(* IEC 61131-3 sources: plc_simulator/services/codesys/POUs (part 9) *)

(* ---- STC_FB_Calibrate.st ---- *)
(* ============================================================
   STC_FB_Calibrate — Teaching / calibration mode
   ============================================================
   Runs 2 normal tasks per transporter to measure real lift,
   sink, and travel kinematic parameters.

   Task 1: lift=dry_station, sink=wet_station
     → MeasureMoveTimes records: lift_s[dry], sink_s[wet],
       travel[dry→wet]
     → X velocity profile measured during phase 3.

   Task 2: lift=wet_station, sink=dry_station
     → MeasureMoveTimes records: lift_s[wet], sink_s[dry],
       travel[wet→dry]

   Two tasks give ALL measurements: lift_wet, sink_wet,
   lift_dry, sink_dry, and X kinematics from vel profile.

   Calibration sequence per transporter:
     Step 10-12: Task 1 (dry→wet) + X velocity measurement
     Step 20-22: Task 2 (wet→dry)
     Step 30:    Read results from g_move → g_cal
     Step 40:    Next transporter or cal_step 100

   Global control:
     Step   0: Idle (waiting for cmd=1)
     Step 100: All measurement done (waiting for cmd=2 = Calculate)
     Step 200: Calculating g_move from measured parameters
     Step 999: Complete (waiting for cmd=3 = abort/reset)

   Inputs:
     i_run  — enable (typically init_done)
     i_cmd  — one-shot command: 1=start, 2=calculate, 3=abort

   Outputs:
     o_step   — current cal_step number
     o_tid    — transporter being calibrated
     o_active — TRUE while calibration is running
   ============================================================ *)

FUNCTION_BLOCK STC_FB_Calibrate
VAR_INPUT
  i_run : BOOL;       (* enable — typically init_done *)
  i_cmd : INT;        (* one-shot: 1=start, 2=calculate, 3=abort *)
END_VAR
VAR_OUTPUT
  o_step   : INT;     (* current calibration cal_step *)
  o_tid    : INT;     (* transporter being calibrated *)
  o_active : BOOL;    (* calibration in progress *)
END_VAR
VAR_EXTERNAL CONSTANT
    MAX_Transporters    : INT;
    MIN_StationIndex : INT;
    MAX_StationIndex   : INT;
END_VAR

VAR_EXTERNAL
  g_transporter : ARRAY[1..MAX_Transporters] OF UDT_TransporterStatusType;
  g_sim_trans   : ARRAY[1..MAX_Transporters] OF UDT_JC_SimTransporterType;
  g_station    : ARRAY[MIN_StationIndex..MAX_StationIndex] OF UDT_StationType;
  g_cfg         : ARRAY[1..MAX_Transporters] OF UDT_TransporterType;
  g_cal         : ARRAY[1..MAX_Transporters] OF UDT_JC_CalibrationType;
  g_move        : ARRAY[1..MAX_Transporters] OF UDT_JC_MoveTimesType;
  g_time_s      : LINT;
END_VAR
VAR
  cal_step       : INT := 0;
  tid        : INT := 0;      (* current transporter 1..3 *)
  task_key   : LINT := 0;   (* task_id for issued task *)
  (* X velocity measurement during phase 3 of task 1 *)
  x_meas_ph  : INT := 0;      (* 0=wait 1=accel 2=cruise 3=decel *)
  x_timer    : REAL := 0.0;
  x_prev_v   : REAL := 0.0;
  x_max_v    : REAL := 0.0;
  x_acc_t    : REAL := 0.0;
  x_dec_t    : REAL := 0.0;
  cur_v      : REAL;
  (* Calculation loop variables *)
  ci         : INT;
  cj         : INT;
  dist       : REAL;
  d_acc      : REAL;
  d_dec      : REAL;
  v_peak     : REAL;
  travel_t   : REAL;
  vm         : REAL;
  ta         : REAL;
  td         : REAL;
  (* Helper *)
  next_tid   : INT;
  wet_idx    : INT;
  dry_idx    : INT;
END_VAR

IF NOT i_run THEN
  RETURN;
END_IF;

(* ── Command handling ── *)
IF i_cmd = 1 AND cal_step = 0 THEN
  (* Start calibration — find first active transporter with plan *)
  tid := 0;
  FOR ci := 1 TO MAX_Transporters DO
    IF g_transporter[ci].IsActive AND tid = 0 THEN
      IF g_cal[ci].WetStation > 0 AND g_cal[ci].DryStation > 0 THEN
        tid := ci;
      END_IF;
    END_IF;
  END_FOR;
  IF tid > 0 THEN
    cal_step := 10;
    o_active := TRUE;
  END_IF;
END_IF;

IF i_cmd = 2 AND cal_step = 100 THEN
  (* Calculate g_move from measured parameters *)
  cal_step := 200;
END_IF;

IF i_cmd = 3 THEN
  (* Abort — reset to idle *)
  cal_step := 0;
  tid := 0;
  o_active := FALSE;
END_IF;

(* ================================================================
   STEP 10-12: TASK 1 — lift=dry_station, sink=wet_station
   MeasureMoveTimes records lift_s[dry], sink_s[wet], travel[dry→wet].
   X velocity profile measured during phase 3 (travel dry→wet).
   ================================================================ *)
IF cal_step = 10 THEN
  (* Issue task 1: lift from dry, sink to wet *)
  task_key := g_time_s;
  g_transporter[tid].TaskId := task_key;
  g_transporter[tid].LiftStationTarget := g_cal[tid].DryStation;
  g_transporter[tid].SinkStationTarget := g_cal[tid].WetStation;
  (* Reset X velocity measurement *)
  x_meas_ph := 0;
  x_timer   := 0.0;
  x_prev_v  := 0.0;
  x_max_v   := 0.0;
  x_acc_t   := 0.0;
  x_dec_t   := 0.0;
  cal_step := 11;
END_IF;

IF cal_step = 11 THEN
  (* Wait for task acceptance *)
  IF g_sim_trans[tid].RunningTaskId = task_key THEN
    cal_step := 12;
  END_IF;
END_IF;

IF cal_step = 12 THEN
  cur_v := ABS(DINT_TO_REAL(g_sim_trans[tid].XVelocity));

  (* ── Track X velocity during phase 3 (travel dry→wet) ── *)
  IF g_transporter[tid].Phase = 3 THEN
    IF x_meas_ph = 0 AND cur_v > 0.5 THEN
      (* Acceleration started *)
      x_meas_ph := 1;
      x_timer := 0.02;
      x_prev_v := cur_v;
      x_max_v := cur_v;

    ELSIF x_meas_ph = 1 THEN
      x_timer := x_timer + 0.02;
      IF cur_v > x_max_v THEN
        x_max_v := cur_v;
      END_IF;
      IF cur_v <= x_prev_v THEN
        (* Velocity stopped increasing → reached v_max *)
        x_acc_t := x_timer - 0.02;
        x_meas_ph := 2;
        x_timer := 0.0;
      END_IF;
      x_prev_v := cur_v;

    ELSIF x_meas_ph = 2 THEN
      (* Cruising — wait for deceleration *)
      IF cur_v < x_max_v - 1.0 THEN
        x_meas_ph := 3;
        x_timer := 0.02;
      END_IF;

    ELSIF x_meas_ph = 3 THEN
      x_timer := x_timer + 0.02;
    END_IF;
  END_IF;

  (* ── Phase 3 ended or phase 4 reached: store X results ── *)
  IF g_transporter[tid].Phase >= 4 AND x_meas_ph >= 1 THEN
    IF x_meas_ph = 3 THEN
      x_dec_t := x_timer;
    END_IF;
    g_cal[tid].XAccelTime  := REAL_TO_INT(x_acc_t * 10.0);
    g_cal[tid].XDecelTime  := REAL_TO_INT(x_dec_t * 10.0);
    g_cal[tid].XMaxSpeed := REAL_TO_DINT(x_max_v);
    (* Don't re-enter — set meas_ph to done *)
    x_meas_ph := 99;
  END_IF;

  (* ── Wait for full task completion (phase returns to 0) ── *)
  IF g_transporter[tid].Phase = 0 AND x_meas_ph >= 99 THEN
    cal_step := 20;
  END_IF;
END_IF;

(* ================================================================
   STEP 20-22: TASK 2 — lift=wet_station, sink=dry_station
   MeasureMoveTimes records lift_s[wet], sink_s[dry], travel[wet→dry].
   ================================================================ *)
IF cal_step = 20 THEN
  (* Issue task 2: lift from wet, sink to dry *)
  task_key := g_time_s + LINT#1;
  g_transporter[tid].TaskId := task_key;
  g_transporter[tid].LiftStationTarget := g_cal[tid].WetStation;
  g_transporter[tid].SinkStationTarget := g_cal[tid].DryStation;
  cal_step := 21;
END_IF;

IF cal_step = 21 THEN
  IF g_sim_trans[tid].RunningTaskId = task_key THEN
    cal_step := 22;
  END_IF;
END_IF;

IF cal_step = 22 THEN
  (* Wait for task completion *)
  IF g_transporter[tid].Phase = 0 THEN
    cal_step := 30;
  END_IF;
END_IF;

(* ================================================================
   STEP 30: READ RESULTS FROM g_move → g_cal
   MeasureMoveTimes has recorded all 4 lift/sink times into g_move.
   ================================================================ *)
IF cal_step = 30 THEN
  wet_idx := g_cal[tid].WetStation - 100;
  dry_idx := g_cal[tid].DryStation - 100;

  IF wet_idx >= 1 AND wet_idx <= 25 THEN
    g_cal[tid].LiftWetTime := g_move[tid].LiftTime[wet_idx];
    g_cal[tid].SinkWetTime := g_move[tid].SinkTime[wet_idx];
  END_IF;

  IF dry_idx >= 1 AND dry_idx <= 25 THEN
    g_cal[tid].LiftDryTime := g_move[tid].LiftTime[dry_idx];
    g_cal[tid].SinkDryTime := g_move[tid].SinkTime[dry_idx];
  END_IF;

  cal_step := 40;
END_IF;

(* ================================================================
   STEP 40: TRANSPORTER DONE — advance to next or finish
   ================================================================ *)
IF cal_step = 40 THEN
  (* Find next active transporter after current tid with plan *)
  next_tid := 0;
  FOR ci := tid + 1 TO MAX_Transporters DO
    IF g_transporter[ci].IsActive AND next_tid = 0 THEN
      IF g_cal[ci].WetStation > 0 AND g_cal[ci].DryStation > 0 THEN
        next_tid := ci;
      END_IF;
    END_IF;
  END_FOR;

  IF next_tid > 0 THEN
    (* Calibrate next transporter *)
    tid := next_tid;
    cal_step := 10;
  ELSE
    (* All transporters done — measurement complete *)
    cal_step := 100;
  END_IF;
END_IF;

(* ================================================================
   STEP 200: CALCULATE g_move FROM MEASURED PARAMETERS
   For each active transporter with calibration data:
     - Copy lift/sink wet times to all wet stations
     - Copy lift/sink dry times to all dry stations
     - Calculate all station-to-station travel times using
       measured v_max, t_acc, t_dec and station distances
   ================================================================ *)
IF cal_step = 200 THEN
  FOR ci := 1 TO MAX_Transporters DO
    IF g_transporter[ci].IsActive AND g_cal[ci].XMaxSpeed > 0 THEN

      vm := DINT_TO_REAL(g_cal[ci].XMaxSpeed);
      ta := INT_TO_REAL(g_cal[ci].XAccelTime) / 10.0;
      td := INT_TO_REAL(g_cal[ci].XDecelTime) / 10.0;

      (* --- Fill lift_s and sink_s per station type --- *)
      FOR cj := 1 TO 25 DO
        IF g_station[100 + cj].TankId <> 0 THEN
          IF g_station[100 + cj].DryWet = 1 THEN
            (* Wet station *)
            g_move[ci].LiftTime[cj] := g_cal[ci].LiftWetTime;
            g_move[ci].SinkTime[cj] := g_cal[ci].SinkWetTime;
          ELSE
            (* Dry station *)
            g_move[ci].LiftTime[cj] := g_cal[ci].LiftDryTime;
            g_move[ci].SinkTime[cj] := g_cal[ci].SinkDryTime;
          END_IF;
        END_IF;
      END_FOR;

      (* --- Calculate all travel times from kinematics --- *)
      (* d_acc = 0.5 * v_max * t_acc (distance during acceleration)
         d_dec = 0.5 * v_max * t_dec (distance during deceleration)
         If dist >= d_acc + d_dec:
           travel = t_acc + (dist - d_acc - d_dec) / v_max + t_dec
         Else (triangle profile):
           v_peak = SQRT(2 * dist * v_max / (t_acc + t_dec))
           travel = v_peak * (t_acc + t_dec) / v_max *)
      d_acc := 0.5 * vm * ta;
      d_dec := 0.5 * vm * td;

      FOR cj := 1 TO 25 DO
        IF g_station[100 + cj].TankId <> 0 THEN
          FOR wet_idx := 1 TO 25 DO
            IF g_station[100 + wet_idx].TankId <> 0 THEN
              IF cj = wet_idx THEN
                g_move[ci].Travel[cj].ToTime[wet_idx] := 0;
              ELSE
                dist := ABS(DINT_TO_REAL(g_station[100 + cj].XPosition - g_station[100 + wet_idx].XPosition));
                IF dist < 1.0 THEN
                  g_move[ci].Travel[cj].ToTime[wet_idx] := 0;
                ELSIF dist >= (d_acc + d_dec) THEN
                  (* Full trapezoidal profile *)
                  travel_t := ta + (dist - d_acc - d_dec) / vm + td;
                  g_move[ci].Travel[cj].ToTime[wet_idx] := REAL_TO_INT(travel_t * 10.0);
                ELSE
                  (* Triangle profile — cannot reach full speed *)
                  IF (ta + td) > 0.0 THEN
                    v_peak := SQRT(2.0 * dist * vm / (ta + td));
                    travel_t := v_peak * (ta + td) / vm;
                    g_move[ci].Travel[cj].ToTime[wet_idx] := REAL_TO_INT(travel_t * 10.0);
                  ELSE
                    g_move[ci].Travel[cj].ToTime[wet_idx] := 0;
                  END_IF;
                END_IF;
              END_IF;
            END_IF;
          END_FOR;
        END_IF;
      END_FOR;

    END_IF;
  END_FOR;

  cal_step := 999;
END_IF;

(* ── Update outputs ── *)
o_step := cal_step;
o_tid  := tid;
IF cal_step > 0 AND cal_step < 999 THEN
  o_active := TRUE;
ELSIF cal_step = 999 THEN
  o_active := FALSE;
ELSE
  o_active := FALSE;
END_IF;

END_FUNCTION_BLOCK

(* ---- STC_FB_ClearTaskQueues.st ---- *)
(* ============================================================
   STC_FB_ClearTaskQueues — Zero-out all transporter task queues
   ============================================================
   Clears count and all 9 fields of each slot in g_task[1..3].

   Replaces 2× identical clear loops in:
     TSK_FB_Scheduler (phase 2000)
     DEP_FB_Scheduler (phase 1020)
   ============================================================ *)

FUNCTION_BLOCK STC_FB_ClearTaskQueues
VAR_EXTERNAL CONSTANT
    MAX_Transporters : INT;
    MAX_Units        : INT;
    MAX_TASK_QUEUE   : INT;
END_VAR

VAR_EXTERNAL
  g_task : ARRAY[1..MAX_Transporters] OF UDT_JC_TskQueueType;
END_VAR
VAR
  ti : INT;
  qi : INT;
END_VAR

FOR ti := 1 TO MAX_Transporters DO
  g_task[ti].Count := 0;
  FOR qi := 1 TO MAX_TASK_QUEUE DO
    g_task[ti].Queue[qi].Unit         := 0;
    g_task[ti].Queue[qi].Stage        := 0;
    g_task[ti].Queue[qi].LiftStationTarget := 0;
    g_task[ti].Queue[qi].SinkStationTarget := 0;
    g_task[ti].Queue[qi].StartTime   := 0;
    g_task[ti].Queue[qi].FinishTime  := 0;
    g_task[ti].Queue[qi].CalcTime    := 0;
    g_task[ti].Queue[qi].MinTime     := 0;
    g_task[ti].Queue[qi].MaxTime     := 0;
  END_FOR;
END_FOR;

END_FUNCTION_BLOCK

(* ---- STC_FB_CollectActiveBatches.st ---- *)
(* ============================================================
   STC_FB_CollectActiveBatches — Filter active batches to list
   ============================================================
   Scans g_batch[1..10] and collects unit indices matching
   mode-specific conditions into an output list.

   Common conditions for both modes:
     unit.Status  = USED (1)
     unit.Target  = TO_NONE (0)
     batch.prog_id = g_program[ui].ProgramId  (valid program)

   Mode:
     i_mode = 0 — active (in-production) batches:
                   batch.state = IN_PROCESS (1)
                   batch.CurStage >= 0 AND <= 99
     i_mode = 1 — waiting batches:
                   Direct lookup: g_station_loc[114].UnitId
                   Only station 114 can hold a waiting batch.

   Replaces 3× duplicated collection loops in:
     TSK_FB_Scheduler (phase 1, active batches)
     DEP_FB_Scheduler (phase 100, active + waiting batches)
   ============================================================ *)

FUNCTION_BLOCK STC_FB_CollectActiveBatches
VAR_INPUT
  i_mode : INT;    (* 0 = all active, 1 = waiting only *)
END_VAR
VAR_EXTERNAL CONSTANT
    MAX_Units : INT;
    MAX_StationIndex : INT;
END_VAR
VAR_EXTERNAL
  g_batch       : ARRAY[1..MAX_Units] OF UDT_BatchType;
  g_unit        : ARRAY[1..MAX_Units] OF UDT_UnitType;
  g_program     : ARRAY[1..MAX_Units] OF UDT_TreatmentProgramType;
  g_station_loc : ARRAY[1..MAX_StationIndex] OF UDT_UnitLocation;
END_VAR
VAR_OUTPUT
  o_list  : ARRAY[1..MAX_Units] OF INT;  (* unit indices *)
  o_count : INT;
END_VAR
VAR
  ui : INT;
END_VAR

o_count := 0;
FOR ui := 1 TO MAX_Units DO
  o_list[ui] := 0;
END_FOR;

IF i_mode = 1 THEN
  (* ── Waiting batch: direct lookup at station 114 ── *)
  ui := g_station_loc[114].UnitId;
  IF ui >= 1 AND ui <= MAX_Units THEN
    IF g_unit[ui].Status = 1
       AND g_unit[ui].Target = 0
       AND g_batch[ui].State = 0
       AND g_batch[ui].ProgId = g_program[ui].ProgramId
       AND g_program[ui].ProgramId > 0 THEN
      o_count := 1;
      o_list[1] := ui;
    END_IF;
  END_IF;
  RETURN;
END_IF;

(* ── Mode 0: active batches — loop ── *)
FOR ui := 1 TO MAX_Units DO
  IF g_unit[ui].Status = 1
     AND g_unit[ui].Target = 0
     AND g_batch[ui].ProgId = g_program[ui].ProgramId
     AND g_program[ui].ProgramId > 0 THEN

    IF g_batch[ui].State = 1
       AND g_batch[ui].CurStage >= 0
       AND g_batch[ui].CurStage <= 99 THEN
      o_count := o_count + 1;
      o_list[o_count] := ui;
    END_IF;
  END_IF;
END_FOR;

END_FUNCTION_BLOCK

(* ---- STC_FB_DispatchTask.st ---- *)
(* ============================================================
   STC_FB_DispatchTask — Validate and dispatch tasks to transporters
   ============================================================
   Called every PLC scan from MainScheduler (before TSK/DEP).
   For each idle transporter with queued tasks:

     1. Skip if transporter not idle (phase <> 0) or queue empty
     2. Time check: is start_time close enough?
        travel_time_to_lift + 3s >= time_until_start → proceed
     3. Sink station free check:
        a) Original sink free → use it
        b) Not free → search alternative parallel stations
           (from g_program[].Steps[] or g_ntt[] for stage=0)
        c) Pick the station with oldest change_time (longest empty)
        d) No free alternative → skip, don't dispatch
     4. Conflict check: no other active transporter targeting
        same lift or sink station
     5. Dispatch: write task_id, lift_station, sink_station
        to g_transporter → RunTasks picks it up

   Used by: STC_FB_MainScheduler
   ============================================================ *)

FUNCTION_BLOCK STC_FB_DispatchTask
VAR_EXTERNAL CONSTANT
    MAX_Transporters    : INT;
    MAX_Units           : INT;
    MAX_STATIONS_PER_STEP       : INT;
    MAX_STEPS_PER_PROGRAM          : INT;
    MIN_StationIndex : INT;
    MAX_StationIndex   : INT;
END_VAR
VAR_EXTERNAL
  g_transporter : ARRAY[1..MAX_Transporters] OF UDT_TransporterStatusType;
  g_sim_trans   : ARRAY[1..MAX_Transporters] OF UDT_JC_SimTransporterType;
  g_task        : ARRAY[1..MAX_Transporters] OF UDT_JC_TskQueueType;
  g_station     : ARRAY[MIN_StationIndex..MAX_StationIndex] OF UDT_StationType;
  g_station_loc : ARRAY[1..MAX_StationIndex] OF UDT_UnitLocation;
  g_unit        : ARRAY[1..MAX_Units] OF UDT_UnitType;
  g_program     : ARRAY[1..MAX_Units] OF UDT_TreatmentProgramType;
  g_ntt         : ARRAY[1..MAX_Transporters] OF UDT_JC_NttTransporterType;
  g_batch       : ARRAY[1..MAX_Units] OF UDT_BatchType;
  g_move        : ARRAY[1..MAX_Transporters] OF UDT_JC_MoveTimesType;
  g_cfg         : ARRAY[1..MAX_Transporters] OF UDT_TransporterType;
  g_schedule    : ARRAY[1..MAX_Units] OF UDT_JC_TskScheduleType;
  g_time_s      : LINT;
  g_event_pending       : UDT_JC_EventMsgType;
  g_event_pending_valid : BOOL;
END_VAR
VAR
  ti           : INT;     (* transporter loop *)
  (* Task fields — read from queue[1] to avoid struct copy *)
  t_unit       : INT;
  t_stage      : INT;
  t_lift       : INT;
  t_sink       : INT;
  t_start      : LINT;
  t_finish     : LINT;
  t_calc_time  : DINT;
  (* Time check *)
  travel_s     : REAL;
  margin_s     : LINT;
  from_idx     : INT;
  to_idx       : INT;
  (* Sink search *)
  sink_stn     : INT;
  sink_free    : BOOL;
  best_stn     : INT;
  best_change  : LINT;
  si           : INT;
  cand_stn     : INT;
  cand_free    : BOOL;
  uj           : INT;
  tgt          : INT;
  ntt_idx      : INT;     (* resolved NTT index (buffer 6/7/8) *)
  ntt_cnt      : INT;
  ntt_fb_cnt   : INT;
  (* Conflict check *)
  conflict     : BOOL;
  cj           : INT;
  task_min     : INT;     (* min station of our proposed task *)
  task_max     : INT;     (* max station of our proposed task *)
  (* Queue position loop *)
  qi           : INT;
  (* Shift-down after dispatch *)
  sh           : INT;
  (* Transfer time for batch progress bar *)
  xfer_total   : REAL;
  (* Program stage number for event *)
  prog_stage   : INT;
END_VAR

FOR ti := 1 TO MAX_Transporters DO

  (* ── 1. Skip if not idle or queue empty ── *)
  IF g_transporter[ti].Phase = 0 AND g_task[ti].Count >= 1 THEN

    (* Try each queue position — skip blocked tasks, dispatch first feasible *)
    FOR qi := 1 TO g_task[ti].Count DO

    (* Read task fields from queue position qi *)
    t_unit      := g_task[ti].Queue[qi].Unit;
    t_stage     := g_task[ti].Queue[qi].Stage;  (* schedule index *)
    t_lift      := g_task[ti].Queue[qi].LiftStationTarget;
    t_sink      := g_task[ti].Queue[qi].SinkStationTarget;
    t_start     := g_task[ti].Queue[qi].StartTime;
    t_finish    := g_task[ti].Queue[qi].FinishTime;
    t_calc_time := g_task[ti].Queue[qi].CalcTime;

    (* Convert schedule index → program stage number for g_program access *)
    prog_stage := 0;
    IF t_unit >= 1 AND t_unit <= MAX_Units THEN
      IF t_stage >= 1 AND t_stage <= g_schedule[t_unit].StageCount THEN
        prog_stage := g_schedule[t_unit].Stages[t_stage].ProgramStage;
      END_IF;
    END_IF;

    (* ── 1b. Lift station unit check — unit must be AT the lift station ── *)
    (* Don't dispatch if unit is not present at the pickup station *)
    IF t_unit >= 1 AND t_unit <= MAX_Units
       AND g_unit[t_unit].location = t_lift THEN

    (* ── 2. Time check ── *)
    travel_s := 0.0;
    IF g_transporter[ti].CurrentStation > 0 AND t_lift > 0
       AND g_transporter[ti].CurrentStation <> t_lift THEN
      from_idx := g_transporter[ti].CurrentStation - 100;
      to_idx   := t_lift - 100;
      IF from_idx >= 1 AND from_idx <= 30 AND to_idx >= 1 AND to_idx <= 30 THEN
        travel_s := INT_TO_REAL(g_move[ti].Travel[from_idx].ToTime[to_idx]) / 10.0;
      END_IF;
    END_IF;

    margin_s := t_start - g_time_s;

    IF margin_s <= REAL_TO_LINT(travel_s) + 3 THEN

      (* ── 3. Sink station free check ── *)
      sink_stn := t_sink;
      sink_free := FALSE;

      IF sink_stn >= MIN_StationIndex AND sink_stn <= MAX_StationIndex THEN
        sink_free := TRUE;
        FOR uj := 1 TO MAX_Units DO
          IF g_unit[uj].location = sink_stn AND g_unit[uj].Status = 1 THEN
            sink_free := FALSE;
          END_IF;
        END_FOR;
      END_IF;

      IF NOT sink_free THEN
        (* Search alternative parallel stations *)
        best_stn := 0;
        best_change := LINT#2000000000;

        IF prog_stage >= 1 AND prog_stage <= MAX_STEPS_PER_PROGRAM
           AND t_unit >= 1 AND t_unit <= MAX_Units THEN
          (* Treatment task — look in g_program for parallel stations *)
          FOR si := 0 TO MAX_STATIONS_PER_STEP - 1 DO
            cand_stn := g_program[t_unit].Steps[prog_stage].Stations[si];
            IF cand_stn > 0 AND cand_stn <> t_sink THEN
              IF cand_stn >= MIN_StationIndex AND cand_stn <= MAX_StationIndex THEN
                cand_free := TRUE;
                FOR uj := 1 TO MAX_Units DO
                  IF g_unit[uj].location = cand_stn AND g_unit[uj].Status = 1 THEN
                    cand_free := FALSE;
                  END_IF;
                END_FOR;
                IF cand_free THEN
                  IF g_station_loc[cand_stn].ChangeTime < best_change THEN
                    best_change := g_station_loc[cand_stn].ChangeTime;
                    best_stn := cand_stn;
                  END_IF;
                END_IF;
              END_IF;
            END_IF;
          END_FOR;

        ELSIF prog_stage = 0 AND t_unit >= 1 AND t_unit <= MAX_Units THEN
          (* No-treatment task — look in g_ntt for alternatives *)
          tgt := g_unit[t_unit].Target;
          IF tgt >= 1 AND tgt <= 5 THEN
            (* Resolve buffer NTT index like NoTreatment does *)
            IF tgt = 2 THEN
              IF g_batch[t_unit].BatchCode = 0 THEN
                ntt_idx := 6;
              ELSIF g_batch[t_unit].State = 2 THEN
                ntt_idx := 8;
              ELSE
                ntt_idx := 7;
              END_IF;
            ELSE
              ntt_idx := tgt;
            END_IF;
            (* Check primary stations *)
            ntt_cnt := g_ntt[ti].Target[ntt_idx].StationCount;
            FOR si := 1 TO ntt_cnt DO
              IF si <= MAX_STATIONS_PER_STEP THEN
                cand_stn := g_ntt[ti].Target[ntt_idx].Stations[si];
                IF cand_stn > 0 AND cand_stn <> t_sink THEN
                  IF cand_stn >= MIN_StationIndex AND cand_stn <= MAX_StationIndex THEN
                    cand_free := TRUE;
                    FOR uj := 1 TO MAX_Units DO
                      IF g_unit[uj].location = cand_stn AND g_unit[uj].Status = 1 THEN
                        cand_free := FALSE;
                      END_IF;
                    END_FOR;
                    IF cand_free THEN
                      IF g_station_loc[cand_stn].ChangeTime < best_change THEN
                        best_change := g_station_loc[cand_stn].ChangeTime;
                        best_stn := cand_stn;
                      END_IF;
                    END_IF;
                  END_IF;
                END_IF;
              END_IF;
            END_FOR;
            (* Check fallback stations *)
            ntt_fb_cnt := g_ntt[ti].Target[ntt_idx].FallbackCount;
            FOR si := 1 TO ntt_fb_cnt DO
              IF si <= MAX_STATIONS_PER_STEP THEN
                cand_stn := g_ntt[ti].Target[ntt_idx].FallbackStations[si];
                IF cand_stn > 0 AND cand_stn <> t_sink THEN
                  IF cand_stn >= MIN_StationIndex AND cand_stn <= MAX_StationIndex THEN
                    cand_free := TRUE;
                    FOR uj := 1 TO MAX_Units DO
                      IF g_unit[uj].location = cand_stn AND g_unit[uj].Status = 1 THEN
                        cand_free := FALSE;
                      END_IF;
                    END_FOR;
                    IF cand_free THEN
                      IF g_station_loc[cand_stn].ChangeTime < best_change THEN
                        best_change := g_station_loc[cand_stn].ChangeTime;
                        best_stn := cand_stn;
                      END_IF;
                    END_IF;
                  END_IF;
                END_IF;
              END_IF;
            END_FOR;
          END_IF;
        END_IF;

        IF best_stn > 0 THEN
          sink_stn := best_stn;
          sink_free := TRUE;
        END_IF;
      END_IF;  (* NOT sink_free *)

      IF sink_free THEN

        (* ── 4. Conflict check ── *)
        (* Check against other transporters' ACTIVE tasks (phase>0).
           Two rules:
           a) T2's entire task (lift AND sink) is inside our task
              range [task_min..task_max] → conflict.
              Example: our 114→101 range [101,114]
                T2 114→113: both in [101,114] → conflict
                T2 114→117: 117 outside     → no conflict (going away)
           b) T2 delivers (sink) to one of our exact stations
              from outside our range → conflict.
              Example: T2 120→114, 114 is our lift → conflict *)
        conflict := FALSE;

        IF t_lift <= sink_stn THEN
          task_min := t_lift;
          task_max := sink_stn;
        ELSE
          task_min := sink_stn;
          task_max := t_lift;
        END_IF;

        FOR cj := 1 TO MAX_Transporters DO
          IF cj <> ti AND g_transporter[cj].Phase > 0 THEN

            (* a) T2's entire active task inside our range → conflict *)
            IF g_transporter[cj].LiftStationTarget >= task_min
               AND g_transporter[cj].LiftStationTarget <= task_max
               AND g_transporter[cj].SinkStationTarget >= task_min
               AND g_transporter[cj].SinkStationTarget <= task_max THEN
              conflict := TRUE;
            END_IF;

            (* b) T2 delivers to one of our exact stations → conflict *)
            IF g_transporter[cj].SinkStationTarget = t_lift
               OR g_transporter[cj].SinkStationTarget = sink_stn THEN
              conflict := TRUE;
            END_IF;

          END_IF;
        END_FOR;

        IF NOT conflict THEN
          (* ── 5. Dispatch: assign task to transporter ── *)
          g_transporter[ti].TaskId      := t_start;
          g_transporter[ti].LiftStationTarget := t_lift;
          g_transporter[ti].SinkStationTarget := sink_stn;
          g_station_loc[ti].UnitId      := t_unit;
          g_sim_trans[ti].TreatmentTime := t_calc_time;
          g_sim_trans[ti].MinTime := g_task[ti].Queue[qi].MinTime;
          g_sim_trans[ti].MaxTime := g_task[ti].Queue[qi].MaxTime;
          g_sim_trans[ti].NttPrimary := g_task[ti].Queue[qi].NttPrimary;
          g_transporter[ti].TaskRemainingTime := t_calc_time;
          g_transporter[ti].TaskFinishTime := t_finish;  (* absolute arrival time at sink station *)

          (* ── Emit TASK_DISPATCHED event (msg_type=1) ── *)
          (* Compute transfer time for xfer_total field *)
          xfer_total := STC_CalcTransferTime(
            i_from_stn            := t_lift,
            i_to_stn              := sink_stn,
            i_move                := g_move[ti],
            i_from_dropping_x10   := g_station[t_lift].DrippingTime,
            i_to_device_delay_x10 := g_station[sink_stn].DeviceDelay,
            i_drip_tray_delay_x10 := g_cfg[ti].DripTrayDelay
          );
          IF xfer_total < 1.0 THEN
            xfer_total := INT_TO_REAL(ABS(sink_stn - t_lift)) * 8.0;
          END_IF;
          IF xfer_total < 5.0 THEN xfer_total := 60.0; END_IF;
          IF NOT g_event_pending_valid THEN
            g_event_pending.MsgType := 1;
            g_event_pending.TsHi := LINT_TO_INT(g_time_s / LINT#65536);
            g_event_pending.TsLo := LINT_TO_INT(g_time_s MOD LINT#65536);
            g_event_pending.Payload[1]  := LINT_TO_INT(t_start / LINT#65536);   (* TaskId_Hi *)
            g_event_pending.Payload[2]  := LINT_TO_INT(t_start MOD LINT#65536);  (* TaskId_Lo *)
            g_event_pending.Payload[3]  := ti;
            g_event_pending.Payload[4]  := t_unit;
            g_event_pending.Payload[5]  := t_lift;
            g_event_pending.Payload[6]  := sink_stn;
            prog_stage := g_batch[t_unit].CurStage;
            g_event_pending.Payload[7]  := prog_stage;  (* treatment program stage number *)
            g_event_pending.Payload[8]  := g_batch[t_unit].BatchCode;
            g_event_pending.Payload[9]  := DINT_TO_INT(t_calc_time);
            g_event_pending.Payload[10] := DINT_TO_INT(g_task[ti].Queue[qi].MinTime);
            g_event_pending.Payload[11] := DINT_TO_INT(g_task[ti].Queue[qi].MaxTime);
            g_event_pending.Payload[12] := REAL_TO_INT(xfer_total);
            g_event_pending_valid := TRUE;
          END_IF;

          (* Copy station-specific timing from config *)
          IF t_lift >= MIN_StationIndex AND t_lift <= MAX_StationIndex THEN
            g_transporter[ti].DrippingTime := g_station[t_lift].DrippingTime;
            g_sim_trans[ti].LiftDeviceDelay := g_station[t_lift].DeviceDelay;
          END_IF;
          IF sink_stn >= MIN_StationIndex AND sink_stn <= MAX_StationIndex THEN
            g_sim_trans[ti].SinkDeviceDelay := g_station[sink_stn].DeviceDelay;
          END_IF;

          (* Shift queue: remove position qi, move rest up *)
          FOR sh := qi + 1 TO g_task[ti].Count DO
            g_task[ti].Queue[sh - 1] := g_task[ti].Queue[sh];
          END_FOR;
          (* Clear last slot *)
          g_task[ti].Queue[g_task[ti].Count].Unit := 0;
          g_task[ti].Queue[g_task[ti].Count].Stage := 0;
          g_task[ti].Queue[g_task[ti].Count].LiftStationTarget := 0;
          g_task[ti].Queue[g_task[ti].Count].SinkStationTarget := 0;
          g_task[ti].Queue[g_task[ti].Count].StartTime := 0;
          g_task[ti].Queue[g_task[ti].Count].FinishTime := 0;
          g_task[ti].Queue[g_task[ti].Count].CalcTime := 0;
          g_task[ti].Queue[g_task[ti].Count].MinTime := 0;
          g_task[ti].Queue[g_task[ti].Count].MaxTime := 0;
          g_task[ti].Count := g_task[ti].Count - 1;
          EXIT;  (* dispatched — stop searching this queue *)

        END_IF;  (* NOT conflict *)

      END_IF;  (* sink_free *)

    END_IF;  (* time check *)

    END_IF;  (* unit at lift station *)

    END_FOR;  (* qi — try next queue position *)

  END_IF;  (* idle + queue *)

END_FOR;

END_FUNCTION_BLOCK

(* ---- STC_FB_EventQueue.st ---- *)
(* ============================================================
   STC_FB_EventQueue — Event message queue handler (OPC UA)
   ============================================================
   Manages a circular 10-slot event queue (g_event).

   - enqueue: caller writes msg fields to g_event_pending,
     then sets g_event_pending_valid := TRUE.
     This FB picks it up and adds to queue.
   - dequeue: Gateway reads g_event.Buffer[Head] directly
     via OPC UA, then writes g_event_ack_seq to acknowledge.
     PLC sees ack match → advance head, count--.

   Called every PLC scan from plc_prg (always, not gated by
   scheduler turn).

   OPC UA handshake:
     PLC:    g_event.Count, g_event.Head, g_event.Buffer[] → readable via OPC UA
     Gateway: g_event_ack_seq → writable via OPC UA
     When g_event_ack_seq = g_event.Buffer[Head].Seq: message consumed → next.
   ============================================================ *)

FUNCTION_BLOCK STC_FB_EventQueue
VAR_EXTERNAL
  g_event               : UDT_JC_EventQueueType;
  g_event_pending       : UDT_JC_EventMsgType;
  g_event_pending_valid : BOOL;
  g_event_ack_seq       : INT;
END_VAR
VAR
  tail : INT;
END_VAR

(* ── 1. Enqueue: pick up pending message if queue not full ── *)
IF g_event_pending_valid AND g_event.Count < 10 THEN
  tail := ((g_event.Head - 1 + g_event.Count) MOD 10) + 1;

  g_event_pending.Seq := g_event.NextSeq;
  g_event.NextSeq := g_event.NextSeq + 1;
  IF g_event.NextSeq > 32000 THEN
    g_event.NextSeq := 1;
  END_IF;

  g_event.Buffer[tail] := g_event_pending;
  g_event.Count := g_event.Count + 1;

  g_event_pending_valid := FALSE;
END_IF;

(* ── 2. Dequeue: check gateway ack for head message ── *)
IF g_event.Count > 0 THEN
  IF g_event_ack_seq = g_event.Buffer[g_event.Head].Seq THEN
    g_event.Head := (g_event.Head MOD 10) + 1;
    g_event.Count := g_event.Count - 1;
  END_IF;
END_IF;

END_FUNCTION_BLOCK

(* ---- STC_FB_FindStation.st ---- *)
(* ============================================================
   fb_station_lookup.stn_data → STC_FB_FindStation — Find a station by its number
   ============================================================ *)

FUNCTION_BLOCK STC_FB_FindStation
VAR_INPUT
  station_number : INT;
END_VAR
VAR_OUTPUT
  found           : BOOL;
  idx             : INT;
  x_mm            : DINT;
  skind           : INT;
  device_delay_s  : REAL;
  dropping_time_s : REAL;
END_VAR
VAR_EXTERNAL CONSTANT
    MIN_StationIndex : INT;
    MAX_StationIndex   : INT;
END_VAR
VAR_EXTERNAL
  g_station : ARRAY[MIN_StationIndex..MAX_StationIndex] OF UDT_StationType;
END_VAR
VAR
  stn_data : UDT_StationType;
END_VAR
  (* Direct lookup by station number — no loop needed *)
  IF (station_number >= MIN_StationIndex) AND (station_number <= MAX_StationIndex) THEN
    stn_data := g_station[station_number];
    IF stn_data.TankId <> 0 THEN
      found := TRUE;
      idx := station_number;
      x_mm := stn_data.XPosition;
      skind := stn_data.DryWet;
      device_delay_s := INT_TO_REAL(stn_data.DeviceDelay) / 10.0;
      dropping_time_s := INT_TO_REAL(stn_data.DrippingTime) / 10.0;
      RETURN;
    END_IF;
  END_IF;

  found := FALSE;
  idx := 0;
  x_mm := 0;
  skind := 0;
  device_delay_s := 0.0;
  dropping_time_s := 0.0;
END_FUNCTION_BLOCK

(* ---- STC_FB_FindTransporter.st ---- *)
(* ===========================================================================================
 *  STC_FB_FindTransporter — Find best covering transporter
 *
 *  Company : Galvatek part of the John Cockerill Group
 *  Author  : Jarmo Piipponen
 *  Created : 25.03.2026
 *
 * -------------------------------------------------------------------------------------------
 *  Finds which transporter (1..3) can handle a lift→sink pair
 *  by checking cfg[].TaskArea[] coverage.
 *
 *  When multiple transporters match, scores by:
 *  1. Fewest queued tasks (load balance)
 *  2. Closest last-sink to new lift (travel efficiency)
 *
 *  If iSinkStn = 0, only lift coverage is checked.
 *
 *  NOTE: Kept as FUNCTION_BLOCK because MATIEC cannot handle
 *  ARRAY OF STRUCT as FUNCTION VAR_INPUT parameter.
 *
 *  ------------------------------------------------------------------------------------------
 *
 *  Changes:
 *
 *
 *
 *)

FUNCTION_BLOCK STC_FB_FindTransporter

(* Introduction of Variables ----------------------------------------------------------------*)

VAR_INPUT
  iLiftStn                : INT;     (* lift station number *)
  iSinkStn                : INT;     (* sink station number, 0 = lift-only search *)
END_VAR

VAR_OUTPUT
  oTrans                   : INT;         (* transporter ID 1..3, 0 = not found *)
END_VAR

VAR_EXTERNAL CONSTANT
    MAX_TRANSPORTERS        : INT;
END_VAR

VAR_EXTERNAL
  Transporters                     : ARRAY[0..MAX_TRANSPORTERS] OF UDT_TransporterType;
  Task                    : ARRAY[1..MAX_TRANSPORTERS] OF UDT_JC_TskQueueType;
END_VAR

VAR
  vTi                        : INT;
  vAi                        : INT;
  vArea                      : UDT_TaskAreaType;
  vCanLift                  : BOOL;
  vCanSink                  : BOOL;
  (* Multi-transporter scoring *)
  vCapable                   : ARRAY[1..3] OF INT;   (* vCapable transporter IDs *)
  vCapCount                 : INT;
  vBestIdx                  : INT;
  vBestCount                : INT;
  vBestDist                 : INT;
  vCurCount                 : INT;
  vCurDist                  : INT;
  vLastSink                 : INT;
  vCi                        : INT;
END_VAR

oTrans := 0;
vCapCount := 0;

(* Phase 1: Collect all vCapable transporters *)
FOR vTi := 1 TO MAX_TRANSPORTERS DO
  FOR vAi := 1 TO 4 DO
    IF vCapCount < 3 THEN
      vArea := Transporters[vTi].TaskArea[vAi];
      IF vArea.MinLift > 0 OR vArea.MaxLift > 0 THEN
        vCanLift := (iLiftStn >= vArea.MinLift) AND (iLiftStn <= vArea.MaxLift);
        IF iSinkStn = 0 THEN
          IF vCanLift THEN
            (* Check not already added — nested IF to avoid array bounds on vCapable[0] *)
            IF vCapCount = 0 THEN
              vCapCount := vCapCount + 1;
              vCapable[vCapCount] := vTi;
            ELSIF vCapable[vCapCount] <> vTi THEN
              vCapCount := vCapCount + 1;
              vCapable[vCapCount] := vTi;
            END_IF;
          END_IF;
        ELSE
          vCanSink := (iSinkStn >= vArea.MinSink) AND (iSinkStn <= vArea.MaxSink);
          IF vCanLift AND vCanSink THEN
            IF vCapCount = 0 THEN
              vCapCount := vCapCount + 1;
              vCapable[vCapCount] := vTi;
            ELSIF vCapable[vCapCount] <> vTi THEN
              vCapCount := vCapCount + 1;
              vCapable[vCapCount] := vTi;
            END_IF;
          END_IF;
        END_IF;
      END_IF;
    END_IF;
  END_FOR;
END_FOR;

(* Phase 2: Select best — score by task count then distance *)
IF vCapCount = 0 THEN
  oTrans := 0;
ELSIF vCapCount = 1 THEN
  oTrans := vCapable[1];
ELSE
  (* JS: scored.sort((a,b) => a.count - b.count || a.distFromLastTask - b.distFromLastTask) *)
  vBestIdx := 1;
  vBestCount := Task[vCapable[1]].Count;
  (* Find last sink station for first candidate *)
  vLastSink := 0;
  IF vBestCount > 0 THEN
    vLastSink := Task[vCapable[1]].Queue[vBestCount].SinkStationTarget;
  END_IF;
  IF vLastSink > 0 THEN
    vBestDist := ABS(vLastSink - iLiftStn);
  ELSE
    vBestDist := 0;
  END_IF;

  FOR vCi := 2 TO vCapCount DO
    vCurCount := Task[vCapable[vCi]].Count;
    vLastSink := 0;
    IF vCurCount > 0 THEN
      vLastSink := Task[vCapable[vCi]].Queue[vCurCount].SinkStationTarget;
    END_IF;
    IF vLastSink > 0 THEN
      vCurDist := ABS(vLastSink - iLiftStn);
    ELSE
      vCurDist := 0;
    END_IF;

    IF vCurCount < vBestCount THEN
      vBestIdx := vCi;
      vBestCount := vCurCount;
      vBestDist := vCurDist;
    ELSIF vCurCount = vBestCount AND vCurDist < vBestDist THEN
      vBestIdx := vCi;
      vBestCount := vCurCount;
      vBestDist := vCurDist;
    END_IF;
  END_FOR;

  oTrans := vCapable[vBestIdx];
END_IF;

END_FUNCTION_BLOCK

(* ---- STC_FB_MainScheduler.st ---- *)
(* ===========================================================================================
 *  STC_FB_MainScheduler — Master scheduler orchestrator
 *
 *  Company : Galvatek part of the John Cockerill Group
 *  Author  : Jarmo Piipponen
 *  Created : 25.03.2026
 *
 * -------------------------------------------------------------------------------------------
 *  Manages TSK_FB_Scheduler and DEP_FB_Scheduler calls on
 *  alternating PLC scan cycles. Ensures they never execute
 *  on the same cycle.
 *
 *  Synchronization rules:
 *  1. Normal: alternate TSK_TURN → DEP_TURN → TSK_TURN
 *  2. Skip DEP when TSK is still computing (phase < 10000)
 *  3. Skip DEP when g_dep_pending.Valid = TRUE
 *  4. g_tsk_stable is computed after each TSK call
 *
 *  Turn values: 0=INIT, 1=TSK_TURN, 2=DEP_TURN
 *
 *  ------------------------------------------------------------------------------------------
 *
 *  Changes:
 *
 *
 *
 *)

FUNCTION_BLOCK STC_FB_MainScheduler

(* Introduction of Variables ----------------------------------------------------------------*)

VAR_INPUT
  i_run                     : BOOL;     (* TRUE = run *)
  i_time_s                  : LINT;     (* current absolute time (s), unix seconds *)
END_VAR

VAR_EXTERNAL
  g_tsk_stable              : BOOL;
  g_conflict_resolved       : BOOL;
  g_dep_pending             : UDT_JC_DepPendingWriteType;
  MAX_UNITS                 : INT;
  NOT_PROCESSED             : INT;
  g_batch                   : ARRAY[1..MAX_UNITS] OF UDT_BatchType;
  g_schedule                : ARRAY[1..MAX_UNITS] OF UDT_JC_TskScheduleType;
  g_dep_wk_schedule         : ARRAY[1..MAX_UNITS] OF UDT_JC_TskScheduleType;
  (* Scheduler debug globals — written here, read by Gateway via OPC UA *)
  g_sched_dbg_tsk_phase     : INT;
  g_sched_dbg_dep_phase     : INT;
  g_sched_dbg_turn          : INT;
  g_sched_dbg_skip_cnt      : INT;
  g_sched_dbg_dep_reject_cnt : INT;
  g_sched_dbg_dep_fit_round : INT;
  g_sched_dbg_dep_cur_wait_unit : INT;
  g_sched_dbg_dep_wait_cnt  : INT;
  g_sched_dbg_batch_cnt     : INT;
  g_sched_dbg_tsk_round_ticks : INT;
  g_sched_dbg_dep_round_ticks : INT;
END_VAR

VAR_OUTPUT
  o_tsk_phase               : INT;     (* TSK scheduler phase *)
  o_dep_phase               : INT;     (* DEP scheduler phase *)
  o_turn                    : INT;     (* 1=TSK ran, 2=DEP ran *)
  o_skip_cnt                : INT;     (* DEP skipped count (debug) *)
END_VAR

VAR
  tsk_sched                 : TSK_FB_Scheduler;
  dep_sched                 : DEP_FB_Scheduler;
  twa_calc                  : TWA_FB_CalcLimits;
  (* dispatch — now FC STC_DispatchTask, no instance needed *)
  turn                      : INT := 0;   (* 0=init, 1=TSK, 2=DEP *)
  skip_cnt                  : INT := 0;
  tsk_phase                 : INT := 0;
  ui                        : INT;
END_VAR

IF NOT i_run THEN
  (* Stop both schedulers *)
  tsk_sched(i_run := FALSE, i_time_s := 0);
  dep_sched(i_run := FALSE, i_time_s := 0, i_tsk_phase := 0);
  turn := 0;
  tsk_phase := 0;
  o_tsk_phase := 0;
  o_dep_phase := 0;
  o_turn := 0;
  RETURN;
END_IF;

(* ── Calculate transporter working areas (X-limits) every cycle ── *)
twa_calc();

(* ── Dispatch tasks to idle transporters (every scan) ── *)
STC_DispatchTask();

(* ── Determine this cycle's turn ── *)
IF turn = 0 THEN
  (* First scan: always start with TSK *)
  turn := 1;

ELSIF turn = 1 THEN
  (* Last cycle was TSK → normally DEP's turn *)
  (* But skip DEP if: *)
  (*   a) TSK has not reached READY yet (phase < 10000) *)
  (*   b) pending data waiting for TSK to process *)
  IF tsk_phase < 10000 THEN
    (* TSK still computing — DEP would be blocked at WAIT_STABLE *)
    turn := 1;
    skip_cnt := skip_cnt + 1;
  ELSIF g_dep_pending.Valid THEN
    (* TSK must process pending before DEP continues *)
    turn := 1;
    skip_cnt := skip_cnt + 1;
  ELSE
    turn := 2;
  END_IF;

ELSIF turn = 2 THEN
  (* Last cycle was DEP → TSK's turn.
     DEP now works on sandbox arrays g_dep_wk_xxx, never live globals,
     so TSK can run freely on any cycle. *)
  turn := 1;
END_IF;

(* ── Execute the selected scheduler ── *)
IF turn = 1 THEN
  (* TSK turn *)
  tsk_sched(i_run := TRUE, i_time_s := i_time_s);
  tsk_phase := tsk_sched.o_phase;

  (* JS parity: set stable only when TSK reached READY and conflictResolved; do not clear here *)
    IF (tsk_phase >= 10000) AND g_conflict_resolved THEN
      g_tsk_stable := TRUE;
  END_IF;

ELSIF turn = 2 THEN
  (* DEP turn *)
  dep_sched(
    i_run       := TRUE,
    i_time_s    := i_time_s,
    i_tsk_phase := tsk_phase
  );
END_IF;

(* ── Publish waiting batch schedules from DEP workspace for UI display ── *)
FOR ui := 1 TO MAX_UNITS DO
  IF g_batch[ui].State = NOT_PROCESSED AND g_dep_wk_schedule[ui].StageCount > 0 THEN
    g_schedule[ui] := g_dep_wk_schedule[ui];
  END_IF;
END_FOR;

(* ── Update outputs ── *)
o_tsk_phase := tsk_sched.o_phase;
o_dep_phase := dep_sched.o_phase;
o_turn      := turn;
o_skip_cnt  := skip_cnt;

(* ── Forward to scheduler debug globals (OPC UA readable) ── *)
g_sched_dbg_tsk_phase        := tsk_sched.o_phase;
g_sched_dbg_dep_phase        := dep_sched.o_phase;
g_sched_dbg_turn             := turn;
g_sched_dbg_skip_cnt         := skip_cnt;
g_sched_dbg_dep_reject_cnt   := dep_sched.o_reject_cnt;
g_sched_dbg_dep_fit_round    := dep_sched.o_fit_round;
g_sched_dbg_dep_cur_wait_unit := dep_sched.o_cur_wait_unit;
g_sched_dbg_dep_wait_cnt     := dep_sched.o_wait_cnt;
g_sched_dbg_batch_cnt        := tsk_sched.o_batch_cnt;
g_sched_dbg_tsk_round_ticks  := tsk_sched.o_round_ticks;
g_sched_dbg_dep_round_ticks  := dep_sched.o_round_ticks;

END_FUNCTION_BLOCK

(* ---- STC_FB_MeasureMoveTimes.st ---- *)
(* ============================================================
   FB_TimeMoves → STC_FB_MeasureMoveTimes — Times actual transporter movements
   ============================================================
   Records real lift, sink, and travel times into g_move table
   by observing phase transitions in the transport cycle.
   Used by task scheduling and departure scheduling.

   Phase state machine (from plc_prg.st):
     0 → 1 : X-travel to lift station
     1 → 2 : Lift at station
     2 → 3 : X-travel to sink station
     3 → 4 : Sink at station
     4 → 0 : Cycle complete

   Filtering — only pure mechanical motion is timed:
     Travel (phase 1, 3): timer runs only when ABS(vel_x) > 0.1
       → filters out TWA collision avoidance stops.
     Lift (phase 2): timer runs only during z_stage 2, 3, 4
       → excludes device_delay + dropping_time (stage 1)
         and drip_delay (stage 5).
     Sink (phase 4): timer runs only during z_stage 7, 8
       → excludes device_delay + drip_delay (stage 6).

   Usage in plc_prg.st (one instance per transporter):
     tm1(t_id := 1, phase := g_transporter[1].Phase,
         delta_t := 0.02, vel_x := g_sim_trans[1].XVelocity,
         z_stage := g_sim_trans[1].ZStage,
         lift_stn := g_transporter[1].LiftStationTarget,
         sink_stn := g_transporter[1].SinkStationTarget,
         from_stn := g_transporter[1].CurrentStation);

   Access recorded times:
     travel := g_move[1].Travel[3].ToTime[11];   stn 103 to 111
     lift   := g_move[1].LiftTime[5];             lift at stn 105
     sink   := g_move[2].SinkTime[12];            sink at stn 112
   ============================================================ *)

FUNCTION_BLOCK STC_FB_MeasureMoveTimes
VAR_INPUT
  t_id     : INT;     (* transporter index 1..3 *)
  phase    : INT;     (* current phase 0..4 *)
  delta_t  : REAL;    (* cycle time in seconds *)
  vel_x    : DINT;    (* current X velocity mm/s *)
  z_stage  : INT;     (* current Z motion stage 0..8 *)
  lift_stn : INT;     (* lift station number, e.g. 105 *)
  sink_stn : INT;     (* sink station number, e.g. 112 *)
  from_stn : INT;     (* station before command was given *)
END_VAR
VAR
  prev_phase   : INT := -1;   (* previous phase for edge detection *)
  timer        : REAL := 0.0; (* running timer *)
  travel_from  : INT;         (* index 1..25 for travel source *)
  travel_to    : INT;         (* index 1..25 for travel destination *)
  lift_idx     : INT;         (* index 1..25 for lift station *)
  sink_idx     : INT;         (* index 1..25 for sink station *)
END_VAR
VAR_EXTERNAL CONSTANT
    MAX_Transporters : INT;
END_VAR

VAR_EXTERNAL
  g_sim_trans : ARRAY[1..MAX_Transporters] OF UDT_JC_SimTransporterType;
  g_move : ARRAY[1..MAX_Transporters] OF UDT_JC_MoveTimesType;
END_VAR

(* ---- Phase transition detection ---- *)
IF phase <> prev_phase THEN

  (* -- Save completed measurement and set up next -- *)

  IF prev_phase = 1 AND phase = 2 THEN
    (* Travel to lift complete → save travel time *)
    IF travel_from >= 1 AND travel_from <= 25
       AND travel_to >= 1 AND travel_to <= 25 THEN
      g_move[t_id].Travel[travel_from].ToTime[travel_to] := REAL_TO_INT(timer * 10.0);
    END_IF;
    (* Start timing lift — timer starts at 0, accumulates only in z_stage 2-4 *)
    lift_idx := lift_stn - 100;
    timer := 0.0;

  ELSIF prev_phase = 2 AND phase = 3 THEN
    (* Lift complete → save lift time (pure mechanical Z-motion only) *)
    IF lift_idx >= 1 AND lift_idx <= 25 THEN
      g_move[t_id].LiftTime[lift_idx] := REAL_TO_INT(timer * 10.0);
    END_IF;
    (* Start timing travel to sink *)
    travel_from := lift_stn - 100;
    travel_to := sink_stn - 100;
    timer := 0.0;

  ELSIF prev_phase = 3 AND phase = 4 THEN
    (* Travel to sink complete → save travel time *)
    IF travel_from >= 1 AND travel_from <= 25
       AND travel_to >= 1 AND travel_to <= 25 THEN
      g_move[t_id].Travel[travel_from].ToTime[travel_to] := REAL_TO_INT(timer * 10.0);
    END_IF;
    (* Start timing sink — timer starts at 0, accumulates only in z_stage 7-8 *)
    sink_idx := sink_stn - 100;
    timer := 0.0;

  ELSIF prev_phase = 4 AND phase = 0 THEN
    (* Sink complete → save sink time (pure mechanical Z-motion only) *)
    IF sink_idx >= 1 AND sink_idx <= 25 THEN
      g_move[t_id].SinkTime[sink_idx] := REAL_TO_INT(timer * 10.0);
    END_IF;
    timer := 0.0;

  ELSIF prev_phase = 0 AND phase = 1 THEN
    (* New cycle starting → set up travel-to-lift *)
    travel_from := from_stn - 100;
    travel_to := lift_stn - 100;
    timer := 0.0;

  ELSE
    (* Unexpected transition → just reset *)
    timer := 0.0;
  END_IF;

  prev_phase := phase;

ELSE
  (* ---- No transition: accumulate timer ---- *)

  IF phase = 1 OR phase = 3 THEN
    (* Travel: only count time when actually moving *)
    (* Filters out TWA collision avoidance stops    *)
    IF vel_x <> 0 THEN
      timer := timer + delta_t;
    END_IF;

  ELSIF phase = 2 THEN
    (* Lift: only mechanical Z-motion stages 2-4 *)
    (* Excludes: stage 1 (device_delay + dropping_time), stage 5 (drip_delay) *)
    IF z_stage >= 2 AND z_stage <= 4 THEN
      timer := timer + delta_t;
    END_IF;

  ELSIF phase = 4 THEN
    (* Sink: only mechanical Z-motion stages 7-8 *)
    (* Excludes: stage 6 (device_delay + drip_delay) *)
    IF z_stage >= 7 AND z_stage <= 8 THEN
      timer := timer + delta_t;
    END_IF;
  END_IF;

END_IF;

END_FUNCTION_BLOCK

(* ---- STC_FB_NoTreatmentStates.st ---- *)
(* ==========================================================
   STC_FB_NoTreatmentStates
   ----------------------------------------------------------
   Manages non-treatment target states for all units.

   Structure:
     Pass 0 — SNAPSHOT: read unit/batch/station state once into
              snap[] array. Also detects has_loading flag.
     Section 1 — PROCESSED: mark last-stage units as PROCESSED.
     Section 2 — TO_AVOID: clear occupied next-stage stations.
     Section 3 — TO_LOADING: route one empty unit to loading.
   ========================================================== *)

FUNCTION_BLOCK STC_FB_NoTreatmentStates
  VAR_EXTERNAL CONSTANT
    MAX_Units          : INT;
    MAX_STEPS_PER_PROGRAM         : INT;
    MAX_STATIONS_PER_STEP      : INT;
    MIN_StationIndex : INT;
    MAX_StationIndex  : INT;
    IN_PROCESS         : INT;
    PROCESSED          : INT;
    NOT_USED           : INT;
    TO_NONE            : INT;
    TO_AVOID           : INT;
    TO_LOADING         : INT;
    USED               : INT;
    OP_LOADING           : INT;
    OP_LOADING_UNLOADING : INT;
  END_VAR

  VAR_EXTERNAL
    g_unit             : ARRAY[1..MAX_Units] OF UDT_UnitType;
    g_batch            : ARRAY[1..MAX_Units] OF UDT_BatchType;
    g_program          : ARRAY[1..MAX_Units] OF UDT_TreatmentProgramType;
    g_station          : ARRAY[MIN_StationIndex..MAX_StationIndex] OF UDT_StationType;
    g_station_loc      : ARRAY[1..MAX_StationIndex] OF UDT_UnitLocation;
    g_time_s           : LINT;
    g_production_queue : INT;
  END_VAR

  VAR
    (* Snapshot *)
    snap        : ARRAY[1..MAX_Units] OF UDT_JC_UnitSnapType;
    u           : INT;        (* unit loop index *)
    has_loading : BOOL;       (* any unit already has TO_LOADING *)
    (* Section 1+2 *)
    p           : INT;        (* parallel station loop *)
    next_stn    : INT;        (* next stage station *)
    occ_uid     : INT;        (* unit_id at an occupied station *)
    free_found  : BOOL;       (* any next-stage station is free *)
    avoid_uid   : INT;        (* unit to mark TO_AVOID *)
    (* Section 3 *)
    load_free   : BOOL;       (* a loading station is free *)
    load_uid    : INT;        (* best candidate for TO_LOADING *)
    load_in_buf : BOOL;       (* current candidate is in buffer *)
    stk         : INT;        (* station loop *)
    op          : INT;        (* station operation code *)
  END_VAR

  (* ════════════════════════════════════════════════════════════
     Pass 0 — SNAPSHOT: collect per-unit state in one pass
     ════════════════════════════════════════════════════════════ *)
  has_loading := FALSE;

  FOR u := 1 TO MAX_Units DO
    snap[u].IsActive := g_unit[u].Status <> NOT_USED;
    IF NOT snap[u].IsActive THEN
      CONTINUE;
    END_IF;

    snap[u].Location       := g_unit[u].location;
    snap[u].Target       := g_unit[u].Target;
    snap[u].HasBatch := g_batch[u].BatchCode <> 0;
    snap[u].BatchState    := g_batch[u].State;
    snap[u].CurStage := g_batch[u].CurStage;

    snap[u].OnStation := snap[u].Location >= MIN_StationIndex
                          AND snap[u].Location <= MAX_StationIndex;
    IF snap[u].OnStation THEN
      snap[u].LocationOp    := g_station[snap[u].Location].StationType;
      snap[u].InBuffer := snap[u].LocationOp >= 44 AND snap[u].LocationOp <= 47;
      IF g_station_loc[snap[u].Location].ChangeTime > 0 THEN
        snap[u].Elapsed := g_time_s - g_station_loc[snap[u].Location].ChangeTime;
      ELSE
        snap[u].Elapsed := 0;
      END_IF;
      IF snap[u].CurStage >= 1 THEN
        snap[u].CalTime := g_program[u].Steps[snap[u].CurStage].CalTime;
      ELSE
        snap[u].CalTime := 0;
      END_IF;
    ELSE
      snap[u].LocationOp    := 0;
      snap[u].InBuffer := FALSE;
      snap[u].Elapsed   := 0;
      snap[u].CalTime       := 0;
    END_IF;

    IF snap[u].Target = TO_LOADING THEN
      has_loading := TRUE;
    END_IF;
  END_FOR;

  (* ════════════════════════════════════════════════════════════
     Section 1 — PROCESSED: mark batch done at last treatment stage
     ════════════════════════════════════════════════════════════
     For each IN_PROCESS unit on a station:
       If next stage is empty (stations[1]=0) → last stage.
       If elapsed >= cal_time → set state := PROCESSED. *)
  FOR u := 1 TO MAX_Units DO
    IF NOT snap[u].IsActive OR NOT snap[u].HasBatch THEN
      CONTINUE;
    END_IF;
    IF snap[u].BatchState <> IN_PROCESS OR NOT snap[u].OnStation THEN
      CONTINUE;
    END_IF;
    IF snap[u].CurStage >= 1 AND snap[u].CurStage < MAX_STEPS_PER_PROGRAM THEN
      IF snap[u].CurStage >= g_program[u].StepCount THEN
        IF snap[u].Elapsed > 0 AND snap[u].Elapsed >= DINT_TO_LINT(snap[u].CalTime) THEN
          g_batch[u].State := PROCESSED;
          snap[u].BatchState   := PROCESSED;  (* update snapshot *)
        END_IF;
      END_IF;
    END_IF;
  END_FOR;

  (* ════════════════════════════════════════════════════════════
     Section 2 — TO_AVOID: clear the way to next treatment station
     ════════════════════════════════════════════════════════════
     For each IN_PROCESS unit whose next stage exists:
       Pass 1: check if any next-stage station is free or already
               has a TO_AVOID unit (slot being cleared).
       Pass 2: if all occupied, mark ONE empty-batch TO_NONE unit
               at those stations as TO_AVOID. *)
  FOR u := 1 TO MAX_Units DO
    IF NOT snap[u].IsActive OR NOT snap[u].HasBatch THEN
      CONTINUE;
    END_IF;
    IF snap[u].BatchState <> IN_PROCESS THEN
      CONTINUE;
    END_IF;
    IF snap[u].CurStage < 1 OR snap[u].CurStage >= MAX_STEPS_PER_PROGRAM THEN
      CONTINUE;
    END_IF;
    IF snap[u].CurStage >= g_program[u].StepCount THEN
      CONTINUE;  (* no next stage *)
    END_IF;

    (* — Pass 1: any next-stage station free or being cleared? — *)
    free_found := FALSE;
    avoid_uid  := 0;
    FOR p := 0 TO MAX_STATIONS_PER_STEP - 1 DO
      next_stn := g_program[u].Steps[snap[u].CurStage].Stations[p];
      IF next_stn = 0 THEN
        EXIT;
      END_IF;
      IF next_stn >= MIN_StationIndex AND next_stn <= MAX_StationIndex THEN
        IF g_station_loc[next_stn].UnitId = 0 THEN
          free_found := TRUE;
          EXIT;
        END_IF;
        occ_uid := g_station_loc[next_stn].UnitId;
        IF occ_uid >= 1 AND occ_uid <= MAX_Units THEN
          IF snap[occ_uid].Target = TO_AVOID THEN
            free_found := TRUE;
            EXIT;
          END_IF;
        END_IF;
      END_IF;
    END_FOR;

    (* — Pass 2: all occupied → mark ONE movable unit TO_AVOID — *)
    IF NOT free_found THEN
      FOR p := 0 TO MAX_STATIONS_PER_STEP - 1 DO
        next_stn := g_program[u].Steps[snap[u].CurStage].Stations[p];
        IF next_stn = 0 THEN
          EXIT;
        END_IF;
        IF next_stn >= MIN_StationIndex AND next_stn <= MAX_StationIndex THEN
          occ_uid := g_station_loc[next_stn].UnitId;
          IF occ_uid >= 1 AND occ_uid <= MAX_Units THEN
            IF NOT snap[occ_uid].HasBatch AND snap[occ_uid].Target = TO_NONE THEN
              avoid_uid := occ_uid;
              EXIT;
            END_IF;
          END_IF;
        END_IF;
      END_FOR;

      IF avoid_uid >= 1 THEN
        g_unit[avoid_uid].Target := TO_AVOID;
        snap[avoid_uid].Target     := TO_AVOID;  (* update snapshot *)
      END_IF;
    END_IF;
  END_FOR;

  (* ════════════════════════════════════════════════════════════
     Section 3 — TO_LOADING: route one empty unit to loading station
     ════════════════════════════════════════════════════════════
     When production is active and a loading/loading_unloading station
     is free, find ONE batchless USED unit with TO_NONE target.
     Priority: units NOT in buffer/storage first. *)
  IF g_production_queue = 1 AND NOT has_loading THEN

    (* Check if any loading station is free *)
    load_free := FALSE;
    FOR stk := MIN_StationIndex TO MAX_StationIndex DO
      op := g_station[stk].StationType;
      IF (op = OP_LOADING OR op = OP_LOADING_UNLOADING)
         AND g_station_loc[stk].UnitId = 0 THEN
        load_free := TRUE;
        EXIT;
      END_IF;
    END_FOR;

    IF load_free THEN
      load_uid    := 0;
      load_in_buf := FALSE;
      FOR u := 1 TO MAX_Units DO
        IF snap[u].IsActive AND NOT snap[u].HasBatch
           AND snap[u].Target = TO_NONE AND snap[u].OnStation THEN
          IF snap[u].InBuffer THEN
            IF load_uid = 0 THEN
              load_uid    := u;
              load_in_buf := TRUE;
            END_IF;
          ELSE
            IF load_uid = 0 OR load_in_buf THEN
              load_uid    := u;
              load_in_buf := FALSE;
            END_IF;
          END_IF;
        END_IF;
      END_FOR;

      IF load_uid >= 1 THEN
        g_unit[load_uid].Target := TO_LOADING;
      END_IF;
    END_IF; (* load_free *)

  END_IF; (* production_queue AND NOT has_loading *)

END_FUNCTION_BLOCK

(* ---- STC_FB_ShiftSchedule.st ---- *)
(* ============================================================
   STC_FB_ShiftSchedule — Shift schedule + task times
   ============================================================
   Propagates a time shift through one unit's schedule stages
   AND through all matching tasks in the 3 transporter queues.

   Positive i_amount = DELAY (shift later),
   Negative i_amount = ADVANCE (shift earlier).

   Replaces 4× duplicated propagation code in TSK_FB_Resolve.
   ============================================================ *)

FUNCTION_BLOCK STC_FB_ShiftSchedule
VAR_INPUT
  i_unit       : INT;     (* unit index 1..10 *)
  i_from_stage : INT;     (* propagate from this stage onward *)
  i_amount     : REAL;    (* seconds to shift (+ = later, - = earlier) *)
END_VAR
VAR_EXTERNAL CONSTANT
    MAX_Transporters : INT;
    MAX_Units        : INT;
END_VAR

VAR_EXTERNAL
  g_schedule : ARRAY[1..MAX_Units] OF UDT_JC_TskScheduleType;
  g_task     : ARRAY[1..MAX_Transporters] OF UDT_JC_TskQueueType;
  g_time_s   : LINT;
END_VAR
VAR
  sc       : INT;
  si       : INT;
  qi       : INT;
  ti       : INT;
  duration : LINT;
END_VAR

IF i_unit < 1 OR i_unit > MAX_Units THEN RETURN; END_IF;
IF ABS(i_amount) < 0.001 THEN RETURN; END_IF;

(* ── Shift schedule stages entry/exit times ── *)
sc := g_schedule[i_unit].StageCount;
FOR si := 1 TO sc DO
  IF si >= 1 AND si <= 30
     AND g_schedule[i_unit].Stages[si].ProgramStage >= i_from_stage THEN
    g_schedule[i_unit].Stages[si].EntryTime :=
      g_schedule[i_unit].Stages[si].EntryTime + REAL_TO_LINT(i_amount);
    g_schedule[i_unit].Stages[si].ExitTime :=
      g_schedule[i_unit].Stages[si].ExitTime + REAL_TO_LINT(i_amount);
    (* GAP-3: Past-clamp — don't let EntryTime go before now+1 *)
    IF i_amount < 0.0 AND g_schedule[i_unit].Stages[si].EntryTime < g_time_s + LINT#1 THEN
      g_schedule[i_unit].Stages[si].ExitTime := g_time_s + LINT#1
        + (g_schedule[i_unit].Stages[si].ExitTime - g_schedule[i_unit].Stages[si].EntryTime);
      g_schedule[i_unit].Stages[si].EntryTime := g_time_s + LINT#1;
    END_IF;
  END_IF;
END_FOR;

(* ── Shift matching tasks in all transporter queues ── *)
FOR ti := 1 TO MAX_Transporters DO
  FOR qi := 1 TO g_task[ti].Count DO
    IF g_task[ti].Queue[qi].Unit = i_unit
       AND g_task[ti].Queue[qi].Stage >= i_from_stage THEN
      g_task[ti].Queue[qi].StartTime :=
        g_task[ti].Queue[qi].StartTime + REAL_TO_LINT(i_amount);
      g_task[ti].Queue[qi].FinishTime :=
        g_task[ti].Queue[qi].FinishTime + REAL_TO_LINT(i_amount);
      (* GAP-3: Past-clamp — don't let StartTime go before now+1 *)
      IF i_amount < 0.0 AND g_task[ti].Queue[qi].StartTime < g_time_s + LINT#1 THEN
        duration := g_task[ti].Queue[qi].FinishTime - g_task[ti].Queue[qi].StartTime;
        g_task[ti].Queue[qi].StartTime := g_time_s + LINT#1;
        g_task[ti].Queue[qi].FinishTime := g_time_s + LINT#1 + duration;
      END_IF;
    END_IF;
  END_FOR;
END_FOR;

END_FUNCTION_BLOCK

(* ---- STC_FB_SortTaskQueue.st ---- *)
(* ============================================================
   STC_FB_SortTaskQueue — Insertion sort task queues by priority
   ============================================================
   Sorts one or all transporter task queues in-place using
   insertion sort (stable, O(n²) — fine for n ≤ 10).

   Priority order (matches JS _compareTasksPriority):
     1. EMERGENCY tasks first (overtime ratio > 1.0)
        — both emergency → higher ratio first
     2. Normal tasks: earliest StartTime first

   Overtime ratio = (g_time_s - batch.StartTime) / batch.MaxTime
   Only computed when batch is IN_PROCESS at the task's lift station
   and batch.CurStage matches task.Stage.

   Mode controlled by i_trans:
     0   = sort ALL queues (1..3)
     1-3 = sort only that transporter's queue

   Replaces 3× duplicated insertion sort code in:
     TSK_FB_Scheduler (phase 2200)
     DEP_FB_Scheduler (phase 1020)
     TSK_FB_Analyze   (merge-sort variant — still inline)
   ============================================================ *)

FUNCTION_BLOCK STC_FB_SortTaskQueue
VAR_INPUT
  i_trans : INT;    (* 0 = all, 1..3 = specific transporter *)
END_VAR
VAR_EXTERNAL CONSTANT
    MAX_Transporters : INT;
    MAX_Units        : INT;
END_VAR

VAR_EXTERNAL
  g_task     : ARRAY[1..MAX_Transporters] OF UDT_JC_TskQueueType;
  g_batch    : ARRAY[1..MAX_Units] OF UDT_BatchType;
  g_unit     : ARRAY[1..MAX_Units] OF UDT_UnitType;
  g_schedule : ARRAY[1..MAX_Units] OF UDT_JC_TskScheduleType;
  g_time_s   : LINT;
END_VAR
VAR
  ti         : INT;
  t_start    : INT;
  t_end      : INT;
  ins_i      : INT;
  ins_j      : INT;
  ins_cnt    : INT;
  tmp_task   : UDT_JC_TskTaskType;
  tmp_unit   : INT;
  cur_unit   : INT;
  tmp_ratio  : REAL;
  cur_ratio  : REAL;
  tmp_emerg  : BOOL;
  cur_emerg  : BOOL;
  do_shift   : BOOL;
END_VAR

IF i_trans >= 1 AND i_trans <= 3 THEN
  t_start := i_trans;
  t_end   := i_trans;
ELSE
  t_start := 1;
  t_end   := 3;
END_IF;

FOR ti := t_start TO t_end DO
  ins_cnt := g_task[ti].Count;
  IF ins_cnt >= 2 THEN
    FOR ins_i := 2 TO ins_cnt DO
      tmp_task := g_task[ti].Queue[ins_i];

      (* ── Compute overtime ratio for the task being inserted ── *)
      tmp_ratio := 0.0;
      tmp_unit  := tmp_task.Unit;
      IF tmp_unit >= 1 AND tmp_unit <= MAX_Units THEN
        IF g_batch[tmp_unit].State = 1                                   (* IN_PROCESS *)
           AND tmp_task.Stage >= 1 THEN
          IF g_batch[tmp_unit].CurStage = tmp_task.Stage
             AND g_unit[tmp_unit].location = tmp_task.LiftStationTarget
             AND g_batch[tmp_unit].StartTime > LINT#0
             AND g_batch[tmp_unit].MaxTime > 0 THEN
            tmp_ratio := LINT_TO_REAL(g_time_s - g_batch[tmp_unit].StartTime)
                         / DINT_TO_REAL(g_batch[tmp_unit].MaxTime);
          END_IF;
        END_IF;
      END_IF;
      tmp_emerg := tmp_ratio > 1.0;

      (* ── Insertion sort with emergency-aware comparator ── *)
      ins_j := 0;
      FOR ins_j := ins_i - 1 TO 1 BY -1 DO
        (* Compute overtime ratio for the element at ins_j *)
        cur_ratio := 0.0;
        cur_unit  := g_task[ti].Queue[ins_j].Unit;
        IF cur_unit >= 1 AND cur_unit <= MAX_Units THEN
          IF g_batch[cur_unit].State = 1
             AND g_task[ti].Queue[ins_j].Stage >= 1 THEN
            IF g_batch[cur_unit].CurStage = g_task[ti].Queue[ins_j].Stage
               AND g_unit[cur_unit].location = g_task[ti].Queue[ins_j].LiftStationTarget
               AND g_batch[cur_unit].StartTime > LINT#0
               AND g_batch[cur_unit].MaxTime > 0 THEN
              cur_ratio := LINT_TO_REAL(g_time_s - g_batch[cur_unit].StartTime)
                           / DINT_TO_REAL(g_batch[cur_unit].MaxTime);
            END_IF;
          END_IF;
        END_IF;
        cur_emerg := cur_ratio > 1.0;

        (* Decide: should Queue[ins_j] shift right to make room for tmp_task? *)
        do_shift := FALSE;
        IF tmp_emerg AND NOT cur_emerg THEN
          (* tmp is emergency, cur is not → tmp goes first *)
          do_shift := TRUE;
        ELSIF tmp_emerg AND cur_emerg THEN
          (* both emergency → higher ratio first *)
          IF tmp_ratio > cur_ratio THEN
            do_shift := TRUE;
          END_IF;
        ELSIF NOT tmp_emerg AND NOT cur_emerg THEN
          (* normal order: earlier StartTime first *)
          IF g_task[ti].Queue[ins_j].StartTime > tmp_task.StartTime THEN
            do_shift := TRUE;
          END_IF;
        (* ELSE: cur is emergency, tmp is not → cur stays, stop *)
        END_IF;

        IF NOT do_shift THEN EXIT; END_IF;

        g_task[ti].Queue[ins_j + 1] := g_task[ti].Queue[ins_j];
      END_FOR;

      g_task[ti].Queue[ins_j + 1] := tmp_task;
    END_FOR;
  END_IF;
END_FOR;

END_FUNCTION_BLOCK

(* ---- STC_FB_TrackMoveTimes.st ---- *)
(* STC_FB_TrackMoveTimes — Record phase transition timestamp and update g_move on completion *)
(* Called from SIM code whenever a transporter phase changes.
   On 4→0 completion, calculates net durations and updates g_move[] with weighted average:
   new = (old * 4 + measured) / 5   (80% old + 20% new) *)
FUNCTION_BLOCK STC_FB_TrackMoveTimes
VAR_INPUT
    i_trans     : INT;   (* transporter index 1..MAX_Transporters *)
    i_prev      : INT;   (* previous phase *)
    i_new       : INT;   (* new phase *)
END_VAR
VAR_TEMP
    t          : INT;
    lift_stn   : INT;
    sink_stn   : INT;
    start_stn  : INT;
    li         : INT;   (* lift station index = stn - 100 *)
    si         : INT;   (* sink station index = stn - 100 *)
    st_i       : INT;   (* start station index = stn - 100 *)
    raw_lift   : INT;   (* measured lift duration ×10 *)
    raw_sink   : INT;   (* measured sink duration ×10 *)
    raw_trav1  : INT;   (* measured travel start→lift ×10 *)
    raw_trav2  : INT;   (* measured travel lift→sink ×10 *)
    drip_x10   : INT;   (* DrippingTime ×10 from lift station *)
    tray_x10   : INT;   (* DripTrayDelay ×10 from transporter config *)
    dev_x10    : INT;   (* DeviceDelay ×10 from sink station *)
END_VAR

t := i_trans;

(* Bounds check *)
IF t < 1 OR t > MAX_Transporters THEN
    RETURN;
END_IF;

CASE i_prev OF
    0: (* 0→1 : siirto nostoasemalle alkaa *)
        IF i_new = 1 THEN
            g_actual_move[t].StartStation := g_transporter[t].CurrentStation;
            g_actual_move[t].LiftStation  := g_transporter[t].LiftStationTarget;
            g_actual_move[t].SinkStation  := g_transporter[t].SinkStationTarget;
            g_actual_move[t].ts0 := g_time_s;
        END_IF;
    1: (* 1→2 : nosto alkaa *)
        IF i_new = 2 THEN
            g_actual_move[t].ts1 := g_time_s;
        END_IF;
    2: (* 2→3 : siirto laskuasemalle alkaa *)
        IF i_new = 3 THEN
            g_actual_move[t].ts2 := g_time_s;
        END_IF;
    3: (* 3→4 : lasku alkaa *)
        IF i_new = 4 THEN
            g_actual_move[t].ts3 := g_time_s;
        END_IF;
    4: (* 4→0 : lasku päättyy — calculate and update g_move *)
        IF i_new = 0 THEN
            g_actual_move[t].ts4 := g_time_s;

            (* Only update if all timestamps are valid *)
            IF g_actual_move[t].ts0 > 0
               AND g_actual_move[t].ts1 > 0
               AND g_actual_move[t].ts2 > 0
               AND g_actual_move[t].ts3 > 0
            THEN
                lift_stn  := g_actual_move[t].LiftStation;
                sink_stn  := g_actual_move[t].SinkStation;
                start_stn := g_actual_move[t].StartStation;
                li   := lift_stn  - 100;
                si   := sink_stn  - 100;
                st_i := start_stn - 100;

                (* Mechanical delays ×10 *)
                drip_x10 := g_station[lift_stn].DrippingTime;
                tray_x10 := g_cfg[t].DripTrayDelay;
                dev_x10  := g_station[sink_stn].DeviceDelay;

                (* Raw durations in ×10 (timestamps are seconds, multiply by 10) *)
                raw_trav1 := LINT_TO_INT((g_actual_move[t].ts1 - g_actual_move[t].ts0) * 10);
                raw_trav2 := LINT_TO_INT((g_actual_move[t].ts3 - g_actual_move[t].ts2) * 10);

                (* Net lift = (ts2-ts1)*10 - DrippingTime - DripTrayDelay *)
                raw_lift := LINT_TO_INT((g_actual_move[t].ts2 - g_actual_move[t].ts1) * 10)
                            - drip_x10 - tray_x10;

                (* Net sink = (ts4-ts3)*10 - DripTrayDelay - DeviceDelay *)
                raw_sink := LINT_TO_INT((g_actual_move[t].ts4 - g_actual_move[t].ts3) * 10)
                            - tray_x10 - dev_x10;

                (* Clamp to minimum 0 *)
                IF raw_lift < 0 THEN raw_lift := 0; END_IF;
                IF raw_sink < 0 THEN raw_sink := 0; END_IF;
                IF raw_trav1 < 0 THEN raw_trav1 := 0; END_IF;
                IF raw_trav2 < 0 THEN raw_trav2 := 0; END_IF;

                (* Bounds check indices *)
                IF li >= 1 AND li <= 30
                   AND si >= 1 AND si <= 30
                   AND st_i >= 1 AND st_i <= 30
                THEN
                    (* Weighted average: new = (old * 4 + measured) / 5 *)

                    (* Lift time at lift station *)
                    g_move[t].LiftTime[li] :=
                        (g_move[t].LiftTime[li] * 4 + raw_lift) / 5;

                    (* Sink time at sink station *)
                    g_move[t].SinkTime[si] :=
                        (g_move[t].SinkTime[si] * 4 + raw_sink) / 5;

                    (* Travel: start → lift (both directions) *)
                    g_move[t].Travel[st_i].ToTime[li] :=
                        (g_move[t].Travel[st_i].ToTime[li] * 4 + raw_trav1) / 5;
                    g_move[t].Travel[li].ToTime[st_i] :=
                        (g_move[t].Travel[li].ToTime[st_i] * 4 + raw_trav1) / 5;

                    (* Travel: lift → sink (both directions) *)
                    g_move[t].Travel[li].ToTime[si] :=
                        (g_move[t].Travel[li].ToTime[si] * 4 + raw_trav2) / 5;
                    g_move[t].Travel[si].ToTime[li] :=
                        (g_move[t].Travel[si].ToTime[li] * 4 + raw_trav2) / 5;
                END_IF;
            END_IF;
        END_IF;
END_CASE;

END_FUNCTION_BLOCK

END_FUNCTION_BLOCK

(* ---- STC_FB_UpdateUnitLocation.st ---- *)
(* ============================================================
   STC_FB_UpdateUnitLocation — Update a unit's location
   ============================================================
   Sets g_unit[i_unit].location to the given new location.
   Location 1..MAX_Transporters = transporter, MIN_StationIndex..MAX_StationIndex = station.
   Updates g_station_loc[location].UnitId + ChangeTime for both.

   When moving to a station (sink / task completion):
     - Advances batch cur_stage if batch is IN_PROCESS
     - Updates batch min_time/max_time/cal_time from treatment program
     - Clears unit target to TO_NONE if target was set (NTT done)
   ============================================================ *)

FUNCTION_BLOCK STC_FB_UpdateUnitLocation
VAR_INPUT
  i_unit        : INT;   (* unit number to update *)
  i_location    : INT;   (* new location: <100 = transporter id, >=100 = station number *)
  i_ntt_primary : INT;   (* 1 = sink is NTT primary → clear target, 0 = don't clear *)
END_VAR
VAR_EXTERNAL CONSTANT
    MAX_Units           : INT;
    MAX_Transporters    : INT;
    MAX_STEPS_PER_PROGRAM          : INT;
    MIN_StationIndex : INT;
    MAX_StationIndex   : INT;
    IN_PROCESS          : INT;
END_VAR
VAR_EXTERNAL
  g_unit        : ARRAY[1..MAX_Units] OF UDT_UnitType;
  g_station     : ARRAY[MIN_StationIndex..MAX_StationIndex] OF UDT_StationType;
  g_station_loc : ARRAY[1..MAX_StationIndex] OF UDT_UnitLocation;
  g_batch       : ARRAY[1..MAX_Units] OF UDT_BatchType;
  g_program     : ARRAY[1..MAX_Units] OF UDT_TreatmentProgramType;
  g_transporter : ARRAY[1..MAX_Transporters] OF UDT_TransporterStatusType;
  g_move        : ARRAY[1..MAX_Transporters] OF UDT_JC_MoveTimesType;
  g_time_s      : LINT;
END_VAR
VAR
  old_loc     : INT;
  new_stg     : INT;
  xfer_total  : REAL;
END_VAR

IF (i_unit >= 1) AND (i_unit <= MAX_Units) THEN
  old_loc := g_unit[i_unit].location;

  (* --- Clear unit_id from old location (unified: transporter or station) --- *)
  IF (old_loc >= 1) AND (old_loc <= MAX_StationIndex) THEN
    g_station_loc[old_loc].UnitId     := 0;
    g_station_loc[old_loc].ChangeTime := g_time_s;
  END_IF;

  (* --- Update unit location --- *)
  g_unit[i_unit].location := i_location;

  (* NOTE: transporter batch times are set directly in SIM_FB_RunTasks
     at LIFT moment, not here — UpdateUnitLocation's transporter block
     was unreliably executing. *)

  (* --- Set unit_id on new location (unified: transporter or station) --- *)
  IF (i_location >= 1) AND (i_location <= MAX_StationIndex) THEN
    g_station_loc[i_location].UnitId     := i_unit;
    g_station_loc[i_location].ChangeTime := g_time_s;

    (* Station-specific: batch stage advance only when landing on a station *)
    IF (i_location >= MIN_StationIndex) THEN

    (* Advance batch stage if unit is USED with an active batch *)
    IF (g_unit[i_unit].Status = 1)  (* USED *)
       AND (g_batch[i_unit].BatchCode <> 0)
       AND (g_batch[i_unit].State = IN_PROCESS)
       AND (g_batch[i_unit].CurStage < MAX_STEPS_PER_PROGRAM) THEN
      g_batch[i_unit].CurStage := g_batch[i_unit].CurStage + 1;

      (* Stamp arrival time on new station — used by CalcSchedule for elapsed calculation *)
      g_batch[i_unit].StartTime := g_time_s;

      (* Update batch treatment times from program for the new stage *)
      IF (g_program[i_unit].ProgramId = g_batch[i_unit].ProgId)
         AND (g_program[i_unit].ProgramId > 0) THEN
        new_stg := g_batch[i_unit].CurStage;
        IF (new_stg >= 1) AND (new_stg <= MAX_STEPS_PER_PROGRAM) THEN
          g_batch[i_unit].MinTime := g_program[i_unit].Steps[new_stg].MinTime;
          g_batch[i_unit].MaxTime := g_program[i_unit].Steps[new_stg].MaxTime;
          g_batch[i_unit].CalTime := g_program[i_unit].Steps[new_stg].CalTime;
        END_IF;
      END_IF;
    END_IF;

    (* NOT_PROCESSED batch on station: clear times so UI shows no progress bar *)
    IF (g_batch[i_unit].BatchCode <> 0)
       AND (g_batch[i_unit].State <> IN_PROCESS) THEN
      g_batch[i_unit].MinTime   := 0;
      g_batch[i_unit].CalTime   := 0;
      g_batch[i_unit].MaxTime   := 32000;  (* ~8.9 h cap, INT max safe *)
      g_batch[i_unit].StartTime := g_time_s;
    END_IF;

    (* Clear unit target ONLY when i_ntt_primary = 1 (primary NTT destination).
       All other cases: keep target so NTT retries primary later. *)
    IF g_unit[i_unit].Target <> 0 AND i_ntt_primary > 0 THEN
      g_unit[i_unit].Target := 0;  (* primary reached → clear *)
    END_IF;

    END_IF; (* i_location >= MIN_StationIndex — station-specific block *)
  END_IF; (* i_location valid *)
END_IF;

END_FUNCTION_BLOCK

(* ---- STC_FindTransporter.st ---- *)
(* ===========================================================================================
 *  STC_FindTransporter — Find best covering transporter
 *
 *  Company : Galvatek part of the John Cockerill Group
 *  Author  : Jarmo Piipponen
 *  Created : 25.03.2026
 *
 * -------------------------------------------------------------------------------------------
 *  Finds which transporter (1..3) can handle a lift→sink pair
 *  by checking cfg[].TaskArea[] coverage.
 *
 *  When multiple transporters match, scores by:
 *  1. Fewest queued tasks (load balance)
 *  2. Closest last-sink to new lift (travel efficiency)
 *
 *  If i_sink_stn = 0, only lift coverage is checked.
 *
 *  NOTE: Kept as FUNCTION_BLOCK because MATIEC cannot handle
 *  ARRAY OF STRUCT as FUNCTION VAR_INPUT parameter.
 *
 *  ------------------------------------------------------------------------------------------
 *
 *  Changes:
 *
 *
 *
 *)

FUNCTION_BLOCK STC_FindTransporter

(* Introduction of Variables ----------------------------------------------------------------*)

VAR_INPUT
  i_lift_stn                : INT;     (* lift station number *)
  i_sink_stn                : INT;     (* sink station number, 0 = lift-only search *)
END_VAR

VAR_OUTPUT
  o_trans                   : INT;         (* transporter ID 1..3, 0 = not found *)
END_VAR

VAR_EXTERNAL CONSTANT
    MAX_TRANSPORTERS        : INT;
END_VAR

VAR_EXTERNAL
  Transporters                     : ARRAY[0..MAX_TRANSPORTERS] OF UDT_TransporterType;
  g_task                    : ARRAY[1..MAX_TRANSPORTERS] OF UDT_JC_TskQueueType;
END_VAR

VAR
  ti                        : INT;
  ai                        : INT;
  area                      : UDT_TaskArea;
  can_lift                  : BOOL;
  can_sink                  : BOOL;
  (* Multi-transporter scoring *)
  capable                   : ARRAY[1..3] OF INT;   (* capable transporter IDs *)
  cap_count                 : INT;
  best_idx                  : INT;
  best_count                : INT;
  best_dist                 : INT;
  cur_count                 : INT;
  cur_dist                  : INT;
  last_sink                 : INT;
  ci                        : INT;
END_VAR

o_trans := 0;
cap_count := 0;

(* Phase 1: Collect all capable transporters *)
FOR ti := 1 TO MAX_TRANSPORTERS DO
  FOR ai := 1 TO 4 DO
    IF cap_count < 3 THEN
      area := Transporters[ti].TaskArea[ai];
      IF area.MinLift > 0 OR area.MaxLift > 0 THEN
        can_lift := (i_lift_stn >= area.MinLift) AND (i_lift_stn <= area.MaxLift);
        IF i_sink_stn = 0 THEN
          IF can_lift THEN
            (* Check not already added — nested IF to avoid array bounds on capable[0] *)
            IF cap_count = 0 THEN
              cap_count := cap_count + 1;
              capable[cap_count] := ti;
            ELSIF capable[cap_count] <> ti THEN
              cap_count := cap_count + 1;
              capable[cap_count] := ti;
            END_IF;
          END_IF;
        ELSE
          can_sink := (i_sink_stn >= area.MinSink) AND (i_sink_stn <= area.MaxSink);
          IF can_lift AND can_sink THEN
            IF cap_count = 0 THEN
              cap_count := cap_count + 1;
              capable[cap_count] := ti;
            ELSIF capable[cap_count] <> ti THEN
              cap_count := cap_count + 1;
              capable[cap_count] := ti;
            END_IF;
          END_IF;
        END_IF;
      END_IF;
    END_IF;
  END_FOR;
END_FOR;

(* Phase 2: Select best — score by task count then distance *)
IF cap_count = 0 THEN
  o_trans := 0;
ELSIF cap_count = 1 THEN
  o_trans := capable[1];
ELSE
  (* JS: scored.sort((a,b) => a.count - b.count || a.distFromLastTask - b.distFromLastTask) *)
  best_idx := 1;
  best_count := g_task[capable[1]].Count;
  (* Find last sink station for first candidate *)
  last_sink := 0;
  IF best_count > 0 THEN
    last_sink := g_task[capable[1]].Queue[best_count].SinkStationTarget;
  END_IF;
  IF last_sink > 0 THEN
    best_dist := ABS(last_sink - i_lift_stn);
  ELSE
    best_dist := 0;
  END_IF;

  FOR ci := 2 TO cap_count DO
    cur_count := g_task[capable[ci]].Count;
    last_sink := 0;
    IF cur_count > 0 THEN
      last_sink := g_task[capable[ci]].Queue[cur_count].SinkStationTarget;
    END_IF;
    IF last_sink > 0 THEN
      cur_dist := ABS(last_sink - i_lift_stn);
    ELSE
      cur_dist := 0;
    END_IF;

    IF cur_count < best_count THEN
      best_idx := ci;
      best_count := cur_count;
      best_dist := cur_dist;
    ELSIF cur_count = best_count AND cur_dist < best_dist THEN
      best_idx := ci;
      best_count := cur_count;
      best_dist := cur_dist;
    END_IF;
  END_FOR;

  o_trans := capable[best_idx];
END_IF;

END_FUNCTION_BLOCK
